KUKA KRL data list: dai_ctrl_library.dat

&ACCESS RVO17
&REL 40
&COMMENT daimler_programcontrol_library
&USER PKL_AST
&PARAM DISKPATH = DAI
&PARAM version = 2.0
DEFDAT  dai_ctrl_library PUBLIC

;FOLD EXTERNAL DECLARATIONS;%{PE}%MKUKATPBASIS,%CEXT,%VCOMMON,%P
;FOLD BASISTECH EXT;%{PE}%MKUKATPBASIS,%CEXT,%VEXT,%P
EXT  BAS (BAS_COMMAND  :IN,REAL  :IN )
DECL INT SUCCESS
;ENDFOLD (BASISTECH EXT)
;FOLD USER EXT;%{E}%MKUKATPUSER,%CEXT,%VEXT,%P
;Make your modifications here



;ENDFOLD (USER EXT)
;ENDFOLD (EXTERNAL DECLARATIONS)


;FOLD GhostOperation

DECL GLOBAL BOOL GhostAllowed=TRUE

DECL GLOBAL CONST INT I_GhostActive=3220
DECL GLOBAL CONST INT I_GhostNonActive=3221
DECL GLOBAL CONST INT O_GhostActive=3220
DECL GLOBAL CONST INT O_GhostAllowed=3221


;ENDFOLD (GhostOperation)

;FOLD HaltPunktEnde_V1.01
;Parametrierung
DECL GLOBAL CONST INT I_HaltNachPunkt=3217
DECL GLOBAL CONST INT O_HaltNachPunktErreicht=3217


INT IntHPE=33
INT CycFlagHPE=33

GLOBAL INT CycFlagWaitForOn=34



DECL GLOBAL BOOL HaltPunktEndeErlaubt=FALSE
DECL GLOBAL BOOL HaltPunktEndeAktiv=TRUE
DECL GLOBAL BOOL HaltPunktEndeOhneHalt=FALSE
DECL GLOBAL INT HPE_OV_PRO_Rett ;Laufzeitvariable:
;ENDFOLD HaltPunktEnde


;
;ENDFOLD (Collstop)


ENDDAT
